END_FUNCTION_BLOCK

// POUs/Engineering/signal processing/SH_T
FUNCTION_BLOCK SH_T
VAR_INPUT
	IN : REAL;
	E : BOOL;
END_VAR
VAR_OUTPUT
	OUT : REAL;
END_VAR


(*
version 1.1	18. oct. 2008
programmer 	hugo
tested by	oscat

this sample and hold module samples an input while en is high.
during the high time of en the output follows in.
the out stays stable until the en goes high again.
*)

IF E THEN out := in; END_IF;



(* revision history
hm	1. sep. 2006	rev 1.0
	original version

hm	18. oct. 2008	rev 1.1
	changed input en to e for compatibility reasons

*)

END_FUNCTION_BLOCK

// POUs/Logic/gate logic/SHL1
FUNCTION SHL1 : DWORD
VAR_INPUT
	IN : DWORD;
	N : INT;
END_VAR
VAR CONSTANT
	temp : DWORD := 16#FFFF_FFFF;
END_VAR

(*
version 1.1	27 dec 2007
programmer 	hugo
tested by		tobias

SHL1 shifts N bits to the left filling the new bits with 1

*)

SHL1 := SHR(temp,32-N) OR SHL(IN,N);


(* revision history
hm	14.9.2007		rev 1.0
	original version

hm	27. dec 2007	rev 1.1
	changed code for better performance

*)

END_FUNCTION

// POUs/Logic/gate logic/SHR1
FUNCTION SHR1 : DWORD
VAR_INPUT
	IN : DWORD;
	N : INT;
END_VAR
VAR CONSTANT
	temp : DWORD := 16#FFFF_FFFF;
END_VAR

(*
version 1.1	27 dec 2007
programmer 	hugo
tested by		tobias

SHR1 shifts N bits to the right filling the new bits with 1

*)

SHR1 := SHL(temp,32-N) OR SHR(IN,N);

(* revision history
hm	14.9.2007		rev 1.0
	original version

hm	27. dec 2007	rev 1.1
	changed code for better performance

*)

END_FUNCTION

// POUs/Logic/FF edge triggered/SHR_4E
FUNCTION_BLOCK SHR_4E
VAR_INPUT
	SET : BOOL;
	D0: BOOL;
	CLK: BOOL;
	RST: BOOL;
END_VAR
VAR_OUTPUT
	Q0: BOOL;
	Q1: BOOL;
	Q2: BOOL;
	Q3: BOOL;
END_VAR
VAR
	trig : R_TRIG;
END_VAR

(*
version 1.1	25. oct. 2008
programmer 	hugo
tested by		tobias

4 bit shift register with reset

*)

(* trig.Q signals a rising edge on clk *)
trig(clk := clk);

IF set OR rst THEN
	Q0 := NOT rst;
	Q1 := Q0;
	Q2 := Q0;
	Q3 := Q0;
ELSIF trig.Q THEN
	Q3 := Q2;
	Q2 := Q1;
	Q1 := Q0;
	Q0 := D0;
END_IF;



(* revision history
hm	4. aug. 2006	rev 1.0
	original version

hm	25. oct. 2008	rev 1.1
	optimized code

*)

END_FUNCTION_BLOCK

// POUs/Logic/FF edge triggered/SHR_4UDE
FUNCTION_BLOCK SHR_4UDE
VAR_INPUT
	SET : BOOL;
	D0: BOOL;
	D3: BOOL;
	CLK: BOOL;
	DN : BOOL;
	RST: BOOL;

END_VAR
VAR_OUTPUT
	Q0: BOOL;
	Q1: BOOL;
	Q2: BOOL;
	Q3: BOOL;
END_VAR
VAR
	trig : R_TRIG;
END_VAR

(*
version 1.2	14. mar. 2009
programmer 	hugo
tested by		tobias

4 bit shift register with reset up / down direction input

*)

(* trig.Q signals a rising edge on clk *)
trig(clk := clk);

IF set OR rst THEN
	Q0 := NOT RST;
	Q1 := Q0;
	Q2 := Q0;
	Q3 := Q0;
ELSIF trig.Q THEN
	IF dn THEN
		Q0 := Q1;
		Q1 := Q2;
		Q2 := Q3;
		Q3 := D3;
	ELSE
		Q3 := Q2;
		Q2 := Q1;
		Q1 := Q0;
		Q0 := D0;
	END_IF;
END_IF;



(* revision history
hm	4. aug. 2006	rev 1.0
	original version

hm	25. oct. 2008	rev 1.1
	optimized code

hm	14. mar. 2009	rev 1.2
	removed double assignments

*)

END_FUNCTION_BLOCK

// POUs/Logic/FF edge triggered/SHR_8PLE
FUNCTION_BLOCK SHR_8PLE
VAR_INPUT
	Din : BOOL;
	Dload : BYTE;
	CLK: BOOL;
	UP: BOOL :=1;
	load : BOOL;
	RST: BOOL;
END_VAR
VAR_OUTPUT
	DOut: BOOL;
END_VAR
VAR
	edge : BOOL :=1;
	register : BYTE;
END_VAR

(*
version 1.0	4 aug 2006
programmer 	hugo
tested by	oscat

8 bit shift register with reset and parallel load
the register can shift up or down
it also has a serial input.
the Din input is on Bit0 for up shift and on bit 7 for down shift
the Dout output is on Bit7 for up shift and on bit 0 for down shift
paralle clock is performed clock synchron while a shift is performed first and then the register is reloaded


*)

(* flankenerkennung clk wird high und edge war high reset ist nicht aktiv und set ist nicht aktiv *)
IF CLK AND edge AND NOT rst THEN
	edge := FALSE;	(* flanke wurde erkannt und weitere flankenerkennung wird verhindert bis edge wieder true ist *)
	(* hier ist der code für das flankenevent *)
	IF UP THEN						(*shift up *)
		register := SHL(register,1);
		register.0 := Din;
		Dout := register.7;
	ELSE								(* shift down *);
		register := SHR(register,1);
		register.7 := Din;
		Dout := register.0;
	END_IF;
	IF load THEN							(* the byte on Din will be loaded if load = true *)
		register := Dload;
		IF up THEN Dout := register.7; ELSE Dout := register.0; END_IF;
	END_IF;
END_IF;
IF NOT clk THEN edge := TRUE; END_IF;	(* sobald clk wieder low wird warten auf nächste flanke *)
IF rst THEN									(* wenn reset aktiv dann ausgang rücksetzen *)
	register := 0;
	Dout := FALSE;
END_IF;

END_FUNCTION_BLOCK

// POUs/Logic/FF edge triggered/SHR_8UDE
FUNCTION_BLOCK SHR_8UDE
VAR_INPUT
	SET : BOOL;
	D0: BOOL;
	D7: BOOL;
	CLK: BOOL;
	DN : BOOL;
	RST: BOOL;
END_VAR
VAR_OUTPUT
	Q0: BOOL;
	Q1: BOOL;
	Q2: BOOL;
	Q3: BOOL;
	Q4: BOOL;
	Q5: BOOL;
	Q6: BOOL;
	Q7: BOOL;
END_VAR
VAR
	trig : R_TRIG;
END_VAR

(*
version 1.2	14. mar. 2009
programmer 	hugo
tested by		tobias

8 bit shift register with reset


*)

(* trig.Q signals a rising edge on clk *)
trig(clk := clk);

IF set OR rst THEN
	Q0 := NOT RST;
	Q1 := Q0;
	Q2 := Q0;
	Q3 := Q0;
	Q4 := Q0;
	Q5 := Q0;
	Q6 := Q0;
	Q7 := Q0;
ELSIF trig.Q THEN
	IF dn THEN
		Q0 := Q1;
		Q1 := Q2;
		Q2 := Q3;
		Q3 := Q4;
		Q4 := Q5;
		Q5 := Q6;
		Q6 := Q7;
		Q7 := D7;
	ELSE
		Q7 := Q6;
		Q6 := Q5;
		Q5 := Q4;
		Q4 := Q3;
		Q3 := Q2;
		Q2 := Q1;
		Q1 := Q0;
		Q0 := D0;
	END_IF;
END_IF;



(* revision history
hm	4. aug. 2006	rev 1.0
	original version

hm	25. oct. 2008	rev 1.1
	optimized code

hm	14. mar. 2009	rev 1.2
	removed double assignments

*)

END_FUNCTION_BLOCK

// POUs/Mathematical/SIGMOID
FUNCTION SIGMOID : REAL
VAR_INPUT
	X : REAL;
END_VAR


(*
version 1.2	10. mar. 2009
programmer 	hugo
tested by		tobias

this function calculates the sigmoid function

*)

IF X > 20.0 THEN
	SIGMOID := 1.0;
ELSIF x < -85.0 THEN
	SIGMOID := 0.0;
ELSE
	SIGMOID := 1.0 / (1.0 + EXP(-X));
END_IF;


(* revision history
hm	10.12.2007		rev 1.0
	original version

hm	11. mar. 2008		rev 1.1
	extended range of valid inputs to +inv / -inv

hm 10. mar. 2009		rev 1.2
	real constants updated to new systax using dot																																																																																																																																																																																																																																																																																																																																																																																																																																																																																																																																																																																																																																																																																																																																																																																																																																																																																																																																																																																																																																																											

*)

END_FUNCTION

// POUs/Mathematical/SIGN_I
FUNCTION SIGN_I : BOOL
VAR_INPUT
	IN : DINT;
END_VAR


(*
version 1.3	27. oct. 2008
programmer 	hugo
tested by	tobias

this function return true if the integer input is negative

*)

SIGN_I := in.31;

(* revision history
hm 3.3.2007	rev 1.1
	changed method of function for better compatibility to other systems

hm	1.12.2007	rev 1.2
	changed code to improve performance

hm	27. oct. 2008	rev 1.3
	changed type of input to dint

*)

END_FUNCTION

// POUs/Engineering/automation/SIGNAL_4
FUNCTION_BLOCK SIGNAL_4
VAR_INPUT
	IN1 : BOOL;
	IN2 : BOOL;
	IN3 : BOOL;
	IN4 : BOOL;
	TS : TIME;
END_VAR
VAR_INPUT CONSTANT
	S1 : BYTE := 2#1111_1111;
	S2 : BYTE := 2#1111_0000;
	S3 : BYTE := 2#1010_1010;
	S4 : BYTE := 2#1010_0000;
END_VAR
VAR_OUTPUT
	Q : BOOL;
END_VAR
VAR
	sig : SIGNAL;
END_VAR

(*
version 1.0	13 dec 2007
programmer 	hugo
tested by		tobias

this function generates one out of 4 signals specified by bit patterns S1 .. S4.
the selected pattern will be shifted with the step time TS.
In1 has higher priority then In2 which has higher priority then IN3 and in4 has the lowest priority.
ts defaults to 128 ms if not specified.
*)

(* an alarm is present read system time first *)
(* check if an alarm is present if yes set sig to the alarm pattern otherwise exit the routine *)
IF in1 THEN
	sig(in := TRUE, sig := s1, TS := TS);
ELSIF in2 THEN
	sig(in := TRUE, sig := s2, TS := TS);
ELSIF in3 THEN
	sig(in := TRUE, sig := s3, TS := TS);
ELSIF in4 THEN
	sig(in := TRUE, sig := s4, TS := TS);
ELSE
	sig(in := FALSE);
END_IF;

(* set the output *)
Q := sig.Q;


(* revision history
hm	13.12.2007		rev 1.0
	original version

*)

END_FUNCTION_BLOCK

// POUs/Mathematical/SINC
FUNCTION SINC : REAL
VAR_INPUT
	X : REAL;
END_VAR


(*
version 1.2	10. mar. 2009
programmer 	hugo
tested by		tobias

this function calculates the sinc function.

*)

IF X = 0.0 THEN
	SINC := 1.0;
ELSE
	SINC := SIN(x) / x;
END_IF;


(* revision histroy
hm	11. mar. 2008	rev 1.0
	original version

hm	1.12.2007	rev 1.1
	changed code to improove performance

hm 10. mar. 2009	rev 1.2
	real constants updated to new systax using dot																																																																																																																																																																																																																																																																																																																																																																																																																																																																																																																																																																																																																																																																																																																																																																																																																																																																																																																																																																																																																																																											

*)

END_FUNCTION

// POUs/Mathematical/Geometry/SPHERE_V
FUNCTION SPHERE_V : REAL
VAR_INPUT
	rx : REAL;
END_VAR


(*
version 1.2	22. feb 2008
programmer 	hugo
tested by		tobias

sphere_V calculates the Volume of a Sphere


*)

sphere_V := 4.188790205 * Rx * RX * RX;

(* revision histroy
hm	16. oct 2007	rev 1.0
	original version

hm	4. dec 2007		rev 1.1
	changed code for better performance

hm	22. feb 2008		rev 1.2
	changed code for better performance
*)

END_FUNCTION

// POUs/Engineering/automation/SRAMP
FUNCTION_BLOCK SRAMP
VAR_INPUT
	X : REAL;
	A_UP : REAL;
	A_DN :REAL;
	VU_MAX : REAL;
	VD_MAX : REAL;
	LIMIT_HIGH : REAL;
	LIMIT_LOW : REAL;
	RST : BOOL;
END_VAR
VAR_OUTPUT
	Y : REAL;
	V : REAL;
END_VAR
VAR
	cycle_time : TC_S;
	init: BOOL;
END_VAR


(*
	version 1.1	11. mar. 2009
	programmer 	hugo
	tested by		tobias

RAMPS generates output signal which are slew rate and acceleration controlled.

*)

(* read the system_time in microseconds *)
cycle_time();

(* assure range of inputs *)
A_up := MAX(0.0, A_UP);
A_dn := MIN(0.0, A_dn);
VU_max := MAX(0.0, VU_max);
VD_max := MIN(0.0, VD_MAX);

(* calculate the output offset *)
IF rst OR NOT init THEN
	init := TRUE;
	Y := 0.0;
	V := 0.0;
ELSIF X = Y THEN
	v := 0.0;
ELSIF X > Y THEN
	(* output is too low >> ramp up and brake at the end *)
	(* accelerate the speed and limit to vu_max *)
	v := MIN(v + A_UP * cycle_time.TC, vu_max);
	(* calculate the max speed to be able to brake and select the lowest *)
	v := MIN(SQRT((Y-X) * 2.0 * A_DN), v);
	(* calculate the output and obey limits *)
	y := LIMIT(limit_low, y + MIN(v * cycle_time.TC, X-Y), limit_high);
ELSIF X < Y THEN
	(* output is too high >> ramp dn and brake at the end *)
	(* accelerate the speed and limit to vd_max *)
	v := MAX(v + A_DN * cycle_time.TC, vd_max);
	(* calculate the max speed to be able to brake and select the lowest *)
	v := MAX(-SQRT((Y-X) * 2.0 * A_UP), v);
	(* calculate the output and obey limits *)
	y := LIMIT(limit_low, y + MAX(v * cycle_time.TC, X-Y), limit_high);
END_IF;


(* revision history
hm	13. mar. 2008	rev 1.0
	original version

hm	11. mar. 2009	rev 1.1
	real constants updated to new systax using dot																																																																																																																																																																																																																																																																																																																																																																																																																																																																																																																																																																																																																																																																																																																																																																																																																																																																																																																																																																																																																																																											

*)

END_FUNCTION_BLOCK

// POUs/Engineering/measurements/TC_S
FUNCTION_BLOCK TC_S

VAR_OUTPUT
	TC : REAL;
END_VAR
VAR
	init: BOOL;
	tx: DWORD;
	last: DWORD;
END_VAR

(*
	version 1.2	11. mar. 2009
	programmer 	hugo
	tested by		tobias

TC_S delivers the time it was last called on the output TC in seconds.

*)

(* read system timer *)
tx := T_PLC_US();

IF NOT init THEN
	init := TRUE;
	TC := 0.0;
ELSE
	tc := DWORD_TO_REAL(tx - last)*1.0E-6;
END_IF;
last := tx;

(* revision history
hm	13. mar. 2008	rev 1.0
	original version

hm	16. mar 2008	rev 1.1
	added type conversion to avoid warnings under codesys 3.0

hm	11. mar. 2009	rev 1.2
	changed real constants to use dot syntax

*)

END_FUNCTION_BLOCK

// POUs/Logic/memory/STACK_16
FUNCTION_BLOCK STACK_16
VAR_INPUT
	Din : DWORD;
	E : BOOL := TRUE;
	RD : BOOL;
	WD : BOOL;
	RST : BOOL;
END_VAR
VAR_OUTPUT
	Dout : DWORD;
	EMPTY : BOOL := TRUE;
	FULL : BOOL;
END_VAR
VAR
	stack : ARRAY[0..n] OF DWORD;
	pt : INT;
END_VAR
VAR CONSTANT
	n : INT := 15;	(* changing this value will chage the number of stored elements in the fifo *)
END_VAR


(*
version 2.0	25. jul 2009
programmer 	hugo
tested by		oscat

16 Dword STACK memory

*)

IF RST THEN
	(* asynchronous reset for the fifo *)
	pt := 0;
	EMPTY := TRUE;
	FULL := FALSE;
	Dout := 0;
ELSIF E THEN
	IF NOT EMPTY AND RD THEN
		(* read one element *)
		pt := pt - 1;
		Dout := stack[pt];
		EMPTY := pt = 0;
		FULL := FALSE;
	END_IF;
	IF NOT FULL AND WD THEN
		(* write one element *)
		stack[pt] := Din;
		pt := pt + 1;
		FULL := pt > n;
		EMPTY := FALSE;
	END_IF;
END_IF;


(* revision history
hm	4. aug. 2006	rev 1.0
	original version

hm	19. feb 2008	rev 1.1
	performance improvements

hm	17. oct. 2008	rev 1.2
	deleted unnecessary init with 0

hm	27. oct. 2008	rev 1.3
	optimized performance

hm	25. jul 2009	rev 2.0
	changed inputs to allow simultsaneous read and write
*)

END_FUNCTION_BLOCK

// POUs/Logic/memory/STACK_32
FUNCTION_BLOCK STACK_32
VAR_INPUT
	Din : DWORD;
	E : BOOL := TRUE;
	RD : BOOL;
	WD : BOOL;
	RST : BOOL;
END_VAR
VAR_OUTPUT
	Dout : DWORD;
	EMPTY : BOOL := TRUE;
	FULL : BOOL;
END_VAR
VAR
	stack : ARRAY[0..n] OF DWORD;
	pt : INT;
END_VAR
VAR CONSTANT
	n : INT := 31;	(* changing this value will chage the number of stored elements in the fifo *)
END_VAR


(*
version 2.0	25. jul 2009
programmer 	hugo
tested by		oscat

32 Dword STACK memory
*)

IF RST THEN
	(* asynchronous reset for the fifo *)
	pt := 0;
	EMPTY := TRUE;
	FULL := FALSE;
	Dout := 0;
ELSIF E THEN
	IF NOT EMPTY AND RD THEN
		(* read one element *)
		pt := pt - 1;
		Dout := stack[pt];
		EMPTY := pt = 0;
		FULL := FALSE;
	END_IF;
	IF NOT FULL AND WD THEN
		(* write one element *)
		stack[pt] := Din;
		pt := pt + 1;
		FULL := pt > n;
		EMPTY := FALSE;
	END_IF;
END_IF;


(* revision history
hm	4. aug. 2006	rev 1.0
	original version

hm	19. feb 2008	rev 1.1
	performance improvements

hm	17. oct. 2008	rev 1.2
	deleted unnecessary init with 0

ks	27. oct. 2008	rev 1.3
	optimized performance

hm	25. jul 2009	rev 2.0
	changed inputs to allow simultsaneous read and write

*)

END_FUNCTION_BLOCK

// POUs/Engineering/signal processing/STAIR
FUNCTION STAIR : REAL
VAR_INPUT
	X : REAL;
	D : REAL;
END_VAR


(*
version 1.4	10. mar. 2009
programmer 	oscat
tested by		tobias

the function stair converts an anlog input signal to a staircase like output.
D is the step width for the output signal.
if D = 0 then the output follows the input without a chage.
*)

IF D > 0.0 THEN
	STAIR := DINT_TO_REAL(REAL_TO_DINT(X / D)) * D;
ELSE
	STAIR := X;
END_IF;



(* revision history
hm	28 jan 2007		rev 1.0
	original version

hm	27 dec 2007		rev 1.1
	changed code for better performance

hm	6. jan 2008		rev 1.2
	further performance improvement

hm	26. oct. 2008		rev 1.3
	optimized code

hm	10. mar. 2009	rev 1.4
	real constants updated to new systax using dot

*)

END_FUNCTION

// POUs/Engineering/signal processing/STAIR2
FUNCTION_BLOCK STAIR2
VAR_INPUT
	X : REAL;
	D : REAL;
END_VAR
VAR_OUTPUT
	Y: REAL;
END_VAR


(*
version 1.4	10. mar. 2009
programmer 	hugo
tested by		oscat

the function stair2 converts an anlog input signal to a staircase like output.
D is the step width for the output signal. the output will use D as a hysteresis for a stairchange.
if D = 0 then the output follows the input without a chage.
*)

IF D > 0.0 THEN
	IF X >= Y + D OR X <= Y - D THEN Y := FLOOR(X/D) * D; END_IF;
ELSE
	Y := X;
END_IF;



(* revision history
hm	28 jan 2007		rev 1.0
	original version

hm	27. dec 2007	rev 1.1
	changed code for better performance

hm	30. jun. 2008	rev 1.2
	added type conversions to avoid warnings under codesys 3.0																																																																																																																																																																																																																																																											

ks	26. oct. 2008	rev 1.3
	improved code

hm	10. mar. 2009	rev 1.4
	real constants updated to new systax using dot

*)

END_FUNCTION_BLOCK

// POUs/Logic/FF pulse triggered/STORE_8
FUNCTION_BLOCK STORE_8
VAR_INPUT
	Set : BOOL;
	D0,D1, D2, D3, D4, D5, D6, D7 : BOOL;
	Clr : BOOL;
	Rst : BOOL;
END_VAR
VAR_OUTPUT
	Q0, Q1, Q2, Q3, Q4, Q5, Q6, Q7 : BOOL;
END_VAR
VAR
	edge: BOOL;
END_VAR

(*
version 1.2	14. mar. 2009
programmer 	hugo
tested by		oscat

Store_4 stores up to 4 boolean inputs until a reset is clearing the outputs.
the respective output is set with a true at the respective input and stays true until a reset is generated.
a set input is used to set all outputs true at the same time, independent of their inputs.
a clear input is used to reset only the lowest priority of the outputs one at a time.
the lowest priority is q3.

*)

IF rst OR set THEN
	q0 := NOT rst;
	q1 := q0;
	q2 := q0;
	q3 := q0;
	q4 := q0;
	q5 := q0;
	q6 := q0;
	q7 := q0;
ELSE
	IF D0 THEN Q0 := TRUE; END_IF;
	IF D1 THEN Q1 := TRUE; END_IF;
	IF D2 THEN Q2 := TRUE; END_IF;
	IF D3 THEN Q3 := TRUE; END_IF;
	IF D4 THEN Q4 := TRUE; END_IF;
	IF D5 THEN Q5 := TRUE; END_IF;
	IF D6 THEN Q6 := TRUE; END_IF;
	IF D7 THEN Q7 := TRUE; END_IF;

	IF clr AND NOT edge THEN
		IF q0 THEN q0 := FALSE;
		ELSIF q1 THEN q1 := FALSE;
		ELSIF q2 THEN q2 := FALSE;
		ELSIF q3 THEN q3 := FALSE;
		ELSIF q4 THEN q4 := FALSE;
		ELSIF q5 THEN q5 := FALSE;
		ELSIF q6 THEN q6 := FALSE;
		ELSE q7 := FALSE;
		END_IF;
	END_IF;
	edge := clr;
END_IF;


(* revision history
hm	25.12.2007	rev 1.0
	original version

hm	30. oct. 2008	rev 1.1
	optimized performance

hm	14. mar. 2009	rev 1.2
	removed double assignments

*)

END_FUNCTION_BLOCK

// POUs/Logic/gate logic/SWAP_BYTE
FUNCTION SWAP_BYTE : WORD
VAR_INPUT
	IN : WORD;
END_VAR


(*
version 1.0	4 feb 2008
programmer 	hugo
tested by		tobias

This function swaps the high and low byte of the word in.

*)

SWAP_BYTE := ROL(in,8);


(* revision history
hm		4. feb 2008	rev 1.0
	original version

*)

END_FUNCTION

// POUs/Logic/gate logic/SWAP_BYTE2
FUNCTION SWAP_BYTE2 : DWORD
VAR_INPUT
	IN : DWORD;
END_VAR


(*
version 1.0	4 feb 2008
programmer 	hugo
tested by		tobias

This function reverses the byte order in the dword.

*)

Swap_Byte2 := (ROR(in,8) AND 16#FF00FF00) OR (ROL(in,8) AND 16#00FF00FF);

(* revision history
hm		4. feb 2008	rev 1.0
	original version

*)

END_FUNCTION

// POUs/Mathematical/TANC
FUNCTION TANC : REAL
VAR_INPUT
	X : REAL;
END_VAR


(*
version 1.1	10. mar. 2009
programmer 	hugo
tested by		oscat

this function calculates the tanc function.

*)

IF X = 0.0 THEN
	TANC := 1.0;
ELSE
	TANC := TAN(x) / x;
END_IF;


(* revision histroy
hm	23. oct. 2008	rev 1.0
	original version

hm 10. mar. 2009	rev 1.1
	real constants updated to new systax using dot																																																																																																																																																																																																																																																																																																																																																																																																																																																																																																																																																																																																																																																																																																																																																																																																																																																																																																																																																																																																																																																											

*)

END_FUNCTION

// POUs/Mathematical/TANH
FUNCTION TANH : REAL
VAR_INPUT
	X : REAL;
END_VAR


(*
version 1.3	10. mar. 2009
programmer 	hugo
tested by		tobias

this function calculates the tangens hyperbolicus

*)

IF X > 20.0 THEN
	TANH := 1.0;
ELSIF X < -20.0 THEN
	TANH := -1.0;
ELSE
	TANH := 1.0 - 2.0 / (EXP(2.0 * x) + 1.0);
END_IF;


(* revision hisdtory
hm		12.1.2007		rev 1.0
	original version

hm		1.12.2007		rev 1.1
	changed code to improve performance

hm		10. mar 2008	rev 1.2
	corrected an error in formula
	extended range of valid inputs to +/- INV

hm 10. mar. 2009	rev 1.3
	real constants updated to new systax using dot																																																																																																																																																																																																																																																																																																																																																																																																																																																																																																																																																																																																																																																																																																																																																																																																																																																																																																																																																																																																																																																											

*)

END_FUNCTION

// POUs/Engineering/measurements/TC_MS
FUNCTION_BLOCK TC_MS

VAR_OUTPUT
	TC : DWORD;
END_VAR
VAR
	init: BOOL;
	tx: DWORD;
	last: DWORD;
END_VAR

(*
	version 1.0	13 mar 2008
	programmer 	hugo
	tested by		tobias

TC_MS delivers the time it was last called on the output TC in Milliseconds.

*)

(* read system timer *)
tx := T_PLC_MS();

IF NOT init THEN
	init := TRUE;
	TC := 0;
ELSE
	tc := tx - last;
END_IF;
last := tx;

(* revision history
hm		13. mar. 2008	rev 1.0
	original version

*)

END_FUNCTION_BLOCK

// POUs/Engineering/measurements/TC_US
FUNCTION_BLOCK TC_US

VAR_OUTPUT
	TC : DWORD;
END_VAR
VAR
	init: BOOL;
	tx: DWORD;
	last: DWORD;
END_VAR

(*
	version 1.0	13 mar 2008
	programmer 	hugo
	tested by		tobias

TC_US delivers the time it was last called on the output TC in Microseconds.

*)

(* read system timer *)
tx := T_PLC_US();

IF NOT init THEN
	init := TRUE;
	TC := 0;
ELSE
	tc := tx - last;
END_IF;
last := tx;

(* revision history
hm		13. mar. 2008	rev 1.0
	original version

*)

END_FUNCTION_BLOCK

// POUs/Engineering/sensor/TEMP_NI
FUNCTION TEMP_NI : REAL
VAR_INPUT
	Res : REAL;
	R0 : REAL;
END_VAR


(*
version 1.5	10. mar. 2009
programmer 	hugo
tested by		tobias

this function returns the temperature for a nickel sensor in a range from -60..+180 °C *)

TEMP_NI := (SQRT(0.30085225 - 2.66E-3 * (R0 - Res)) - 0.5485) * 751.8796992;


(* revision history

hm 24.1.2007		rev 1.1
	deleted unused variable A, B, C

hm 10.9.2007		rev 1.2
	changed accuracy to 0.02 degrees to improove performace

hm 17. 12 2007	rev 1.3
	improovements for better performance and higher accuracy

hm	6. jan 2008	rev 1.4
	further performance improvement

hm	10. mar. 2009	rev 1.5
	removed nested comments

*)

END_FUNCTION

// POUs/Engineering/sensor/TEMP_NTC
FUNCTION TEMP_NTC : REAL
VAR_INPUT
	RES : REAL;
	RN : REAL;
	B : REAL;
END_VAR


(*
version 1.1	11. mar. 2009
programmer 	hugo
tested by		tobias

this function returs the temperature for a NTC sensor for a range from 0..85 °C.
RN is the resistance at 25 °C and B is a constant for the given sensor.

*)

IF res > 0.0 THEN
	TEMP_NTC := B * 298.15 / (B + LN(RES / RN) * 298.15) -273.15;
END_IF;


(* revision history

hm 30. dec. 2008	rev 1.0
	original version

hm	11. mar. 2009	rev 1.1
	changed real constants to use dot syntax

*)

END_FUNCTION

// POUs/Engineering/sensor/TEMP_PT
FUNCTION TEMP_PT : REAL
VAR_INPUT
	Res : REAL;
	R0 : REAL;
END_VAR
VAR CONSTANT
	A : REAL := 3.9083E-3 ;
	B : REAL := -5.775E-7;
	accuracy : REAL := 0.01;
END_VAR
VAR
	step: REAL := 50.0;
	X: REAL;
	Y: REAL;
	t1: REAL;
	pt : POINTER TO DWORD;
END_VAR

(*
version 1.7	11. mar. 2009
programmer 	hugo
tested by		oscat

this function returs the temperature for a platinum sensor for a range from -200..+850 °C *)

X := A * R0;
Y := B * R0;
IF Res >= R0 THEN
	t1 := X * X - 4.0 * Y * (R0 - Res);
	IF t1 < 0.0 THEN
		TEMP_PT := 10000.0;
	ELSE
		TEMP_PT := (-X + SQRT(t1)) / (2.0 * Y);
	END_IF;
ELSE
	pt := ADR(step);
	(* since the formula cannot be solved this is a successive approximation *)
	TEMP_PT := -100.0;
	WHILE step > accuracy DO
		(* test if result greater or less *)
		IF RES_PT(TEMP_PT, R0) < res THEN TEMP_PT := TEMP_PT + step; ELSE TEMP_PT := TEMP_PT - step; END_IF;
		pt^ := pt^ - 8388608;  (* this is a super fast divide by 2 method for non floating point CPUs *)
		(* the alternative code: step := step * 0.5; *)
	END_WHILE;
END_IF;

(* revision history

rev 1.1 hm 24.1.2007	
	deleted unused variable C

rev 1.2 hm 10.9.2007
	reduced accuracy to 0.02 to shorten execution time

rev 1.3	hm	2. dec 2007
	changed code for better performance

rev	1.4	hm	23. dec 2007
	avoid a negative square root if input values are wrong

rev 1.5 hm	5. jan 2008
	replaced / 2 with * 0.5 for better performance

hm	31. oct. 2008	rev 1.6
	improved performance

hm	11. mar. 2009	rev 1.7
	changed real constants to use dot syntax

*)

END_FUNCTION

// POUs/Engineering/sensor/TEMP_SI
FUNCTION TEMP_SI : REAL
VAR_INPUT
	Res : REAL;
	RS : REAL;
	TS : REAL;
END_VAR


(*
version 1.5	10. mar. 2009
programmer 	hugo
tested by		tobias

this function returs the temperature for a silicon sensor for a range from -60..+180 °C
for example KTY10 RS at TS normally 25 °C
*)

TEMP_SI := (-7.64E-3 + SQRT(Res / RS * 6.64E-5 - 0.803E-5)) * 30120.48193 + TS;



(* revision history

hm 24.1.2007		rev 1.1
	the function would only work for TS = 25, now it works for other values of ts.

hm 10.9.2007		rev 1.2
	changed the function to use successive approcimation to avoid an error generated by a sqrt from a negative result.
	changed accuracy to 0.02 degrees to shorten execution time

hm 17. 12 2007	rev 1.3
	improovements for better performance

hm	6. jan 2008	rev 1.4
	further performance improvement

hm	10. mar. 2009	rev 1.5
	removed nested comments

*)

END_FUNCTION

// POUs/String/TICKER
FUNCTION_BLOCK TICKER

VAR_INPUT
	N : INT;
	PT : TIME;
END_VAR

VAR_IN_OUT
	Text : STRING(STRING_LENGTH);
END_VAR

VAR_OUTPUT
	Display : STRING(STRING_LENGTH);
END_VAR
VAR
	delay : TP;
	step : INT;
END_VAR

(*
version 1.2	29. mar. 2008
programmer 	hugo
tested by		tobias

Ticker sends a substring of text with length N every TD Milliseconds to generate a ticker. 

*)


(* generate next ticker when delay is low *)
IF N < LEN(text) THEN
	IF NOT delay.Q THEN
		(* increase step for next tick *)
		step := step + 1;
		IF step > LEN(text) THEN step := 1; END_IF;
		(* extract dispay from text *)
		display := MID(text, N, step);
		(* set delay timer for next tick *)
		delay(in := TRUE, PT := PT);
	ELSE;
		(* execute delay timer *)
		delay(in := FALSE);
	END_IF;
ELSE
	display := text;
END_IF;
(* revision history
hm	4. dec. 2007	rev 1.0
	original version

hm	15. dec. 2007	rev 1.1
	step now starts at 1 instaed of 0

hm	29. mar. 2008	rev 1.2
	changed STRING to STRING(STRING_LENGTH)
*)

END_FUNCTION_BLOCK

// POUs/Time&Date/TIMECHECK
FUNCTION TIMECHECK : BOOL
VAR_INPUT
	TD : TOD;
	START : TOD;
	STOP : TOD;
END_VAR


(*
version 1.0	19. jul. 2009
programmer 	oscat
tested by		oscat

this function retruns true if the daytime TD is between start and stop and returns true if so.
if you want to generate an event to span over midnight, start timemust be later than the stop time.

*)

IF stop < start THEN
	TIMECHECK := start <= TD OR TD < stop;
ELSE
	TIMECHECK := start <= TD AND TD < stop;
END_IF;



(* revision history
hm 19. jul. 2009	rev 1.0
	original release

*)

END_FUNCTION

// POUs/Logic/generators/TMIN
FUNCTION_BLOCK TMIN
VAR_INPUT
	IN : BOOL;
	PT : TIME;
END_VAR
VAR_OUTPUT
	Q : BOOL;
END_VAR
VAR
	pm : TP;
END_VAR

(*
version 1.0	21. jul. 2008
programmer 	hugo
tested by	oscat

Q of tMIN will follow IN except that it forces a minimum ontime for the output Q.

*)

pm(in := IN, PT := PT);
Q := IN OR pm.Q;


(* revision history
hm	21. jul. 2008	rev 1.0
	original version

*)

END_FUNCTION_BLOCK

// POUs/Logic/generators/TOF_1
FUNCTION_BLOCK TOF_1
VAR_INPUT
	IN : BOOL;
	PT : TIME;
	RST : BOOL;
END_VAR
VAR_OUTPUT
	Q : BOOL;
END_VAR
VAR
	tx : TIME;
	start : TIME;
END_VAR

(*
version 1.0	17. jul. 2008
programmer 	hugo
tested by	oscat

TOF_1 will extend a pulse on input in for PT seconds.
in addition the timer can be cleared asynchronously with rst.
TOF_1 is the same function as TOF from the standard LIB except the asynchronous reset input.

*)

(* read system timer *)
tx := DWORD_TO_TIME(T_PLC_MS());

IF RST THEN
	Q := FALSE;
ELSIF IN THEN
	Q := TRUE;
	start := tx;
ELSIF tx - start >= PT THEN
	Q := FALSE;
END_IF;




(* revision history
hm	17. jul. 2008	rev 1.0
	original version

*)

END_FUNCTION_BLOCK

// POUs/Logic/generators/TONOF
FUNCTION_BLOCK TONOF
VAR_INPUT
	IN : BOOL;
	  T_ON,T_OFF : TIME;
END_VAR
VAR_OUTPUT
	Q : BOOL;
END_VAR
VAR
   X : TON;
   old: BOOL;
   mode: BOOL;
END_VAR

(*
version 1.2	21. jul 2009
programmer 	hugo
tested by		tobias

TONOF generated a TON and TOF Delay for the Input N TON (T1) and TOF (T2) can be configured separately
*)

IF IN XOR old THEN
  X(IN := FALSE, PT := SEL(IN,T_OFF,T_ON));
  mode := IN;
  old := IN;
END_IF;
X(IN := TRUE);
IF X.Q THEN Q := mode;END_IF;

(* revision history
hm	10. dec 2007	rev 1.0
	original version

hm	17. sep. 2007	rev 1.1
	improved performance

hm	21. jul. 2009	rev 1.2
	fixed a timing probelm


*)

END_FUNCTION_BLOCK

// POUs/Logic/generators/TP_1
FUNCTION_BLOCK TP_1
VAR_INPUT
	IN : BOOL;
	PT : TIME;
	RST : BOOL;
END_VAR
VAR_OUTPUT
	Q : BOOL;
END_VAR
VAR
	tx : TIME;
	start : TIME;
	ix : BOOL;
END_VAR

(*
version 1.0	28. jun. 2008
programmer 	hugo
tested by		oscat

TP_1 generates a pulse every time it is calles with in := TRUE.
in addition the timer can be cleared asynchronously with rst.
the timer can be retriggered as often as necessary. it will count PT from the last trigger.

*)

(* read system timer *)
tx := DWORD_TO_TIME(T_PLC_MS());

IF RST THEN
	Q := FALSE;
ELSIF IN AND NOT ix THEN
	Q := TRUE;
	start := tx;
ELSIF tx - start >= PT THEN
	Q := FALSE;
END_IF;

ix:= IN;



(* revision history
hm	28. jun. 2008
	original version

*)

END_FUNCTION_BLOCK

// POUs/Mathematical/Geometry/TRIANGLE_A
FUNCTION TRIANGLE_A : REAL
VAR_INPUT
	S1 : REAL;
	A : REAL;
	S2 : REAL;
	S3 : REAL;
END_VAR


(*
version 1.2	10. mar. 2009
programmer 	hugo
tested by		tobias

triangle_A calculates the Area of a triangle.
if any input is 0 it will be neglected and the are will be calculated from eiter:
two sides and an angle (s1 and S2 and the angle A1) or 3 sides.


*)

IF A = 0.0 THEN
	TRIANGLE_A := SQRT((s1+s2+S3) * (s1+s2-S3) * (S2+S3-S1) * (S3+S1-S2)) * 0.25;
ELSE
	TRIANGLE_A := S1 * S2 * SIN(RAD(A)) * 0.5;
END_IF;

(* revision histroy
hm	16. oct 2007	rev 1.0
	original version

hm	22. feb 2008	rev 1.1
	improved performance

hm	10. mar. 2009	rev 1.2
	changed syntax of real constants to 0.0

*)

END_FUNCTION

// POUs/String/TRIM1
FUNCTION TRIM1 : STRING(STRING_LENGTH)
VAR_INPUT
	str : STRING(STRING_LENGTH);
END_VAR
VAR
	pos: INT;
END_VAR

(*
version 1.2	29. mar. 2008
programmer 	hugo
tested by		tobias

the function replaces all multiple blanks within a string by only one blank.
leading and ending blanks will be deleted

*)

TRIM1 := str;
REPEAT
	pos := FIND(trim1,'  ');
	IF pos > 0 THEN TRIM1 := REPLACE(TRIM1,' ',2,pos); END_IF;
UNTIL pos = 0	END_REPEAT;
(* beginning and ending blanks need to be stripped off *)
IF LEFT(trim1,1) = ' ' THEN trim1 := DELETE(trim1,1,1); END_IF;
IF RIGHT(trim1,1) = ' ' THEN trim1 := DELETE(trim1,1,LEN(trim1)); END_IF;


(* revision histroy
hm	4. feb. 2008    rev 1.0
	original release

hm	20. mar. 2008	rev 1.1
	avoid to call replace with pos = 0 because some systems will produce an error

hm	29. mar. 2008	rev 1.2
	changed STRING to STRING(STRING_LENGTH)
*)

END_FUNCTION

// POUs/String/TRIME
FUNCTION TRIME : STRING(string_length)
VAR_INPUT
	str : STRING(STRING_LENGTH);
END_VAR


(*
version 1.0	28. mar. 2008
programmer 	hugo
tested by	tobias

this function deletes all leading and ending blanks of a string.

*)

TRIME := str;
(* beginning blanks need to be stripped off *)
WHILE LEFT(TRIME,1) = ' ' DO
	TRIME := DELETE(TRIME,1,1);
END_WHILE;

(* ending blanks need to be stripped off *)
WHILE RIGHT(TRIME,1) = ' ' DO
	TRIME := DELETE(TRIME,1,LEN(TRIME));
END_WHILE;


(* revision histroy
hm	28. mar. 2008	rev 1.0
	original release

*)

END_FUNCTION

// POUs/Engineering/automation/TUNE
FUNCTION_BLOCK TUNE
VAR_INPUT
	SET : BOOL;
	SU, SD : BOOL;
	RST : BOOL;
END_VAR
VAR_INPUT CONSTANT
	SS : REAL := 0.1;
	Limit_L : REAL;
	LIMIT_H : REAL := 100.0;
	RST_val : REAL;
	SET_val : REAL := 100.0;
	T1 : TIME := T#500ms;
	T2 : TIME := T#2s;
	S1 : REAL := 2.0;
	S2 : REAL := 10.0;
END_VAR
VAR_OUTPUT
	Y : REAL;
END_VAR
VAR
	tx : DWORD;
	start, start2 : DWORD;
	state : INT;
	in : BOOL;
	step : REAL;
	SPEED : REAL;
	Y_start : REAL;
	Y_start2: REAL;
END_VAR

(*
version 1.2	11. mar. 2009
programmer 	hugo
tested by		tobias

tune generates an output signal which is set by input switches.
up to 4 switsches can be used to tune the signal up or down.

*)

(* read system time *)
tx := T_PLC_MS();

IF rst THEN
	Y := RST_val;
	state := 0;
ELSIF set THEN
	Y := SET_val;
	state := 0;
ELSIF state > 0 THEN
	(* key has been pushed state machine operating *)
	(* first read the correct input *)
	IF state = 1 THEN
		(* step up *)
		in := su;
	ELSE
		(* step down *)
		in := sd;
	END_IF;
	(* check for single step operation *)
	IF NOT in AND tx - start <= TIME_TO_DWORD(T1) THEN
		Y := Y_start + step;
		state := 0;
	(* check if fast ramp needs to be generated *)
	ELSIF in AND tx - start >= TIME_TO_DWORD(T2) THEN
		Y := Y_start2 + DWORD_TO_REAL(tx - start2) * s2 / speed;
	(* check if slow ramp needs to be generated *)
	ELSIF in AND tx - start >= TIME_TO_DWORD(T1) THEN
		Y := Y_start + DWORD_TO_REAL(tx - start - TIME_TO_DWORD(T1)) * S1 / speed;
		start2 := tx;
		Y_start2 := Y;
	ELSIF NOT in THEN
		state := 0;
	END_IF;
ELSIF su THEN
	(* slow step up *)
	state := 1;
	start := tx;
	step := ss;
	speed := 1000.0;
	Y_start := Y;
ELSIF sd THEN
	(* slow step down *)
	state := 2;
	start := tx;
	step := -ss;
	speed := -1000.0;
	Y_start := Y;
END_IF;

(* make sure output does not exceed limits *)
Y := LIMIT(LIMIT_L, Y, LIMIT_H);

(* revision history
hm	3.11.2007		rev 1.0
	original version

hm	16. mar. 2008	rev 1.1
	added type conversions to avoid warnings under codesys 3.0

hm	11. mar. 2009	rev 1.2
	real constants updated to new systax using dot																																																																																																																																																																																																																																																																																																																																																																																																																																																																																																																																																																																																																																																																																																																																																																																																																																																																																																																																																																																																																																																											

*)

END_FUNCTION_BLOCK

// POUs/Engineering/automation/TUNE2
FUNCTION_BLOCK TUNE2
VAR_INPUT
	SET : BOOL;
	SU, SD : BOOL;
	FU, FD : BOOL;
	RST : BOOL;
END_VAR
VAR_INPUT CONSTANT
	SS : REAL := 0.1;
	FS : REAL := 5.0;
	Limit_L : REAL;
	LIMIT_H : REAL := 100.0;
	RST_val : REAL;
	SET_val : REAL := 100.0;
	TR : TIME := T#500ms;
	S1 : REAL := 2.0;
	S2 : REAL := 10.0;
END_VAR
VAR_OUTPUT
	Y : REAL;
END_VAR
VAR
	tx : DWORD;
	start : DWORD;
	state : INT;
	in : BOOL;
	step : REAL;
	SPEED : REAL;
	Y_start : REAL;
END_VAR

(*
version 1.2	11. mar. 2009
programmer 	hugo
tested by		tobias

tune2 generates an output signal which is set by input switches.
up to 4 switsches can be used to tune the signal up or down.

*)

(* read system time *)
tx := T_PLC_MS();

IF rst THEN
	Y := RST_val;
	state := 0;
ELSIF set THEN
	Y := SET_val;
	state := 0;
ELSIF state > 0 THEN
	(* key has been pushed state machine operating *)
	(* first read the correct input *)
	CASE state OF
		1 :	(* slow up *)
			in := su;
		2 :	(* slow down *)
			in := sd;
		3 :	(* fast up *)
			in := fu;
		4 :	(* fast down *)
			in := fd;
	END_CASE;
	(* check for single step operation *)
	IF NOT in AND tx - start <= TIME_TO_DWORD(TR) THEN
		Y := Y_start + step;
		state := 0;
	(* check if ramp needs to be generated *)
	ELSIF in AND tx - start >= TIME_TO_DWORD(TR) THEN
		Y := Y_start + DWORD_TO_REAL(tx - start - TIME_TO_DWORD(TR)) * speed;
	ELSIF NOT in THEN
		state := 0;
	END_IF;
ELSIF su THEN
	(* slow step up *)
	state := 1;
	start := tx;
	step := ss;
	speed := s1 * 1.0E-3;
	Y_start := Y;
ELSIF sd THEN
	(* slow step down *)
	state := 2;
	start := tx;
	step := -ss;
	speed := -s1 * 1.0E-3;
	Y_start := Y;
ELSIF fu THEN
	(* fast step up *)
	state := 3;
	start := tx;
	step := fs;
	speed := s2 * 1.0E-3;
	y_start := Y;
ELSIF fd THEN
	(* fast step down *)
	state := 4;
	start := tx;
	step := -fs;
	speed := -s2 * 1.0E-3;
	y_start := Y;
END_IF;

(* make sure output does not exceed limits *)
Y := LIMIT(LIMIT_L, Y, LIMIT_H);

(* revision history
hm	3.11.2007		rev 1.0
	original version

hm	16. 3. 2008	rev 1.1
	added type conversions to avoid warnings in codesys 3.0
	improved performance

hm	11. mar. 2009	rev 1.2
	real constants updated to new systax using dot																																																																																																																																																																																																																																																																																																																																																																																																																																																																																																																																																																																																																																																																																																																																																																																																																																																																																																																																																																																																																																																											

*)

END_FUNCTION_BLOCK

// POUs/Mathematical/Vektormathematik/V3_ABS
FUNCTION V3_ABS : REAL
VAR_INPUT
	A : Vector_3;
END_VAR


(*
version 1.0	11 dec 2007
programmer 	hugo
tested by		tobias

this function calculates the length of a vectors in a 3 dimensional space

*)

V3_ABS := SQRT(A.X * A.X + A.Y * A.Y + A.Z * A.Z);


(* revision history
hm		11 dec 2007	rev 1.0
	original version

*)

END_FUNCTION

// POUs/Mathematical/Vektormathematik/V3_ADD
FUNCTION V3_ADD : vector_3
VAR_INPUT
	A : Vector_3;
	B : Vector_3;
END_VAR


(*
version 1.0	11 dec 2007
programmer 	hugo
tested by		tobias

this function adds two vectors in a 3 dimensional space

*)

V3_ADD.X := A.X + B.X;
V3_ADD.Y := A.Y + B.Y;
V3_ADD.Z := A.Z + B.Z;



(* revision history
hm		11 dec 2007	rev 1.0
	original version

*)

END_FUNCTION

// POUs/Mathematical/Vektormathematik/V3_ANG
FUNCTION V3_ANG : REAL
VAR_INPUT
	A : Vector_3;
	B : Vector_3;
END_VAR
VAR
	d : REAL;
END_VAR

(*
version 1.1	10. mar. 2009
programmer 	hugo
tested by		tobias

this function calculates the angle between two vectors in a 3 dimensional space

*)

d := V3_ABS(A) * V3_ABS(B);
IF d > 0 THEN
	V3_ANG := ACOS(LIMIT(-1.0, V3_DPRO(A, B) / d,1.0));
END_IF;

(* revision history
hm	11. dec. 2007	rev 1.0
	original version

hm	10. mar. 2009	rev 1.1
	changed syntax of real constants to 0.0

*)

END_FUNCTION

// POUs/Mathematical/Vektormathematik/V3_DPRO
FUNCTION V3_DPRO : REAL
VAR_INPUT
	A : Vector_3;
	B : Vector_3;
END_VAR


(*
version 1.0	11 dec 2007
programmer 	hugo
tested by		tobias

this function calculates the dot product of two vectors in 3 dimensional space

*)

V3_DPRO := A.X * B.X + A.Y * B.Y + A.Z * B.Z;


(* revision history
hm		11 dec 2007	rev 1.0
	original version

*)

END_FUNCTION

// POUs/Mathematical/Vektormathematik/V3_NORM
FUNCTION V3_NORM : vector_3
VAR_INPUT
	A : Vector_3;
END_VAR
VAR
	la: REAL;
END_VAR

(*
version 1.1	10. mar. 2009
programmer 	hugo
tested by		tobias

this function generates a vectors with absolute length 1 from a vector A in a 3 dimensional space

*)

la := V3_ABS(A);
IF la > 0.0 THEN
	V3_NORM := V3_SMUL(A, 1.0 / la);
END_IF;

(* revision history
hm	11 dec 2007	rev 1.0
	original version

hm	10. mar. 2009	rev 1.1
	changed syntax of real constants to 0.0

*)

END_FUNCTION

// POUs/Mathematical/Vektormathematik/V3_SMUL
FUNCTION V3_SMUL : vector_3
VAR_INPUT
	A : Vector_3;
	M : REAL;
END_VAR


(*
version 1.0	11 dec 2007
programmer 	hugo
tested by		tobias

this function multiplies a vectors in a 3 dimensional space with a skalar M

*)

V3_SMUL.X := A.X * M;
V3_SMUL.Y := A.Y * M;
V3_SMUL.Z := A.Z * M;



(* revision history
hm		11 dec 2007	rev 1.0
	original version

*)

END_FUNCTION

// POUs/Mathematical/Vektormathematik/V3_NUL
FUNCTION V3_NUL : BOOL
VAR_INPUT
	A : Vector_3;
END_VAR


(*
version 1.1	10. mar. 2009
programmer 	hugo
tested by		tobias

this function checks if a vectors in a null Vector

*)

V3_NUL := A.X = 0.0 AND A.Y = 0.0 AND A.Z = 0.0;



(* revision history
hm	12 dec 2007	rev 1.0
	original version

hm	10. mar. 2009	rev 1.1
	changed syntax of real constants to 0.0

*)

END_FUNCTION

// POUs/Mathematical/Vektormathematik/V3_PAR
FUNCTION V3_PAR : BOOL
VAR_INPUT
	A : Vector_3;
	B : Vector_3;
END_VAR


(*
version 1.1	10. mar. 2009
programmer 	hugo
tested by		tobias

this function checks if two vectors in a 3 dimensional space are parallel.
which means the two vectors have the same direction

*)

V3_PAR := V3_ABS(V3_XPRO(A, B)) = 0.0;



(* revision history
hm	11 dec 2007	rev 1.0
	original version

hm	10. mar. 2009	rev 1.1
	changed syntax of real constants to 0.0

*)

END_FUNCTION

// POUs/Mathematical/Vektormathematik/V3_XPRO
FUNCTION V3_XPRO : vector_3
VAR_INPUT
	A : Vector_3;
	B : Vector_3;
END_VAR


(*
version 1.0	11 dec 2007
programmer 	hugo
tested by		tobias

this function adds two vectors in a 3 dimensional space

*)

V3_XPRO.X := A.Y * B.Z - A.Z * B.Y;
V3_XPRO.Y := A.Z * B.X - A.X * B.Z;
V3_XPRO.Z := A.X * B.Y - A.Y * B.X;



(* revision history
hm		11 dec 2007	rev 1.0
	original version

*)

END_FUNCTION

// POUs/Mathematical/Vektormathematik/V3_REV
FUNCTION V3_REV : vector_3
VAR_INPUT
	A : Vector_3;
END_VAR


(*
version 1.0	11 dec 2007
programmer 	hugo
tested by		tobias

this function reverses a vector in a 3 dimensional space

*)

V3_REV.X := -A.X;
V3_REV.Y := -A.Y;
V3_REV.Z := -A.Z;



(* revision history
hm		11 dec 2007	rev 1.0
	original version

*)

END_FUNCTION

// POUs/Mathematical/Vektormathematik/V3_SUB
FUNCTION V3_SUB : vector_3
VAR_INPUT
	A : Vector_3;
	B : Vector_3;
END_VAR


(*
version 1.0	11 dec 2007
programmer 	hugo
tested by		tobias

this function subtracts two vectors in a 3 dimensional space
V3_SUB = A - B

*)

V3_SUB.X := A.X - B.X;
V3_SUB.Y := A.Y - B.Y;
V3_SUB.Z := A.Z - B.Z;



(* revision history
hm		11 dec 2007	rev 1.0
	original version

*)

END_FUNCTION

// POUs/Mathematical/Vektormathematik/V3_XANG
FUNCTION V3_XANG : REAL
VAR_INPUT
	A : Vector_3;
END_VAR
VAR
	la: REAL;
END_VAR

(*
version 1.1	10. mar. 2009
programmer 	hugo
tested by		tobias

this function calculates the angle between the X-axis and a vectors in a 3 dimensional space

*)

la := V3_ABS(a);
IF la > 0.0 THEN
	V3_XANG := ACOS(A.X / la);
END_IF;

(* revision history
hm	11 dec 2007	rev 1.0
	original version

hm	10. mar. 2009	rev 1.1
	changed syntax of real constants to 0.0

*)

END_FUNCTION

// POUs/Mathematical/Vektormathematik/V3_YANG
FUNCTION V3_YANG : REAL
VAR_INPUT
	A : Vector_3;
END_VAR
VAR
	la: REAL;
END_VAR

(*
version 1.1	10. mar. 2009
programmer 	hugo
tested by		tobias

this function calculates the angle between the Y-axis and a vectors in a 3 dimensional space

*)

la := V3_ABS(a);
IF la > 0.0 THEN
	V3_YANG := ACOS(A.Y / la);
END_IF;

(* revision history
hm	11 dec 2007	rev 1.0
	original version

hm	10. mar. 2009	rev 1.1
	changed syntax of real constants to 0.0

*)

END_FUNCTION

// POUs/Mathematical/Vektormathematik/V3_ZANG
FUNCTION V3_ZANG : REAL
VAR_INPUT
	A : Vector_3;
END_VAR
VAR
	la: REAL;
END_VAR

(*
version 1.1	10. mar. 2009
programmer 	hugo
tested by		tobias

this function calculates the angle between the Z-axis and a vectors in a 3 dimensional space

*)

la := V3_ABS(a);
IF la > 0.0 THEN
	V3_ZANG := ACOS(A.Z / la);
END_IF;

(* revision history
hm	11 dec 2007	rev 1.0
	original version

hm	10. mar. 2009	rev 1.1
	changed syntax of real constants to 0.0

*)

END_FUNCTION

// POUs/Mathematical/WINDOW2
FUNCTION WINDOW2 : BOOL
VAR_INPUT
	LOW : REAL;
	IN : REAL;
	HIGH : REAL;
END_VAR


(*
	version 1.0	31 oct 2007
	programmer 	hugo
	tested BY	tobias

this checks a signal if the signal is between the upper and lower limit including the two limits
*)

WINDOW2 := IN >= LOW AND IN <= HIGH;


(* revision history
hm	31.10.2007	rev 1.0
	original version

*)

END_FUNCTION

// POUs/Logic/gate logic/WORD_OF_BYTE
FUNCTION WORD_OF_BYTE : WORD
VAR_INPUT
	B1 : BYTE;
	B0 : BYTE;
END_VAR


(*
version 1.4	18. jul. 2009
programmer 	hugo
tested by		tobias

this function creates a word from 2 individual bytes

*)

WORD_OF_BYTE := SHL(BYTE_TO_WORD(B1),8) OR BYTE_TO_WORD(B0);

(* revision history
hm	24. jan 2007	rev 1.0
	original version

hm	2. jan 2008	rev 1.1
	improved performance

hm	19. feb 2008	rev 1.2
	replaced and with or for better compatibility

hm	23. apr. 2008	rev 1.3
	reverse order of inputs to be more logical

hm	18. jul. 2009	rev 1.4
	added type conversions for compatibility reasons

*)

END_FUNCTION

// POUs/Logic/gate logic/WORD_OF_DWORD
FUNCTION WORD_OF_DWORD : WORD
VAR_INPUT
	in : DWORD;
	N : BYTE;
END_VAR


(*
version 1.2	30. oct. 2008
programmer 	hugo
tested by	oscat

this function extracts a single word from the nth position from right (right is lowest byte)
the lower word (starting with Bit0 from in) is selected with N=0.
*)

WORD_OF_DWORD := DWORD_TO_WORD(SHR(in,SHL(n,4)));

(* revision history
hm	17. jan 2007	rev 1.0
	original version

hm	2. jan 2008		rev 1.1
	improved performance

hm	30. oct. 2008	rev 1.2
	improved performance
*)

END_FUNCTION

// POUs/Engineering/signal processing/WORD_TO_RANGE
FUNCTION WORD_TO_RANGE : REAL
VAR_INPUT
	X : WORD;
	low : REAL;
	high : REAL;
END_VAR


(*
version 1.1	10. mar. 2009
programmer 	hugo
tested by		tobias

Word_to_Range converts a Byte into a real between low and high.

*)

WORD_TO_RANGE := (high - low) * WORD_TO_REAL(X) * 0.00001525902189669640 + low;


(* revision history
hm	9. jan 2008	rev 1.0
	original version

hm	10. mar. 2009	rev 1.1
	improved code
*)

END_FUNCTION

// POUs/Time&Date/YEAR_END
FUNCTION YEAR_END : DATE
VAR_INPUT
	y : INT;
END_VAR


(*
version 1.1	24. jan. 2011
programmer 	hugo
tested by	oscat

returs the date of december 31st for the given year  
the function works for dates from 1970 - 2099 

*)

YEAR_END := DWORD_TO_DATE(SHR(INT_TO_DWORD(y) * 1461 - 2876712, 2) * 86400);



(* revision history
hm	15. jun. 2008	rev 1.0
	original version

hm	24. jan 2011	rev 1.1
	improved performance
*)

END_FUNCTION

// POUs/String/LREAL_TO_STRF
FUNCTION LREAL_TO_STRF : STRING(40)
VAR_INPUT
	IN : LREAL;
	N : INT;
	D : STRING(1);
END_VAR
VAR
	O: LREAL;
	i: INT;
END_VAR

(*
version 1.8	2. jan 2012
programmer 	hugo
tested by	oscat

Real_to_strf converts a Real to a fixed length String.
the string will be filles with zeroes to achieve the fixed length N after the decimal separator.
the input parameter specifies the decimal separator to be used in the output string.

*)

(* LIMIT N to 0 .. 17 *)
N := LIMIT(0,N,17);
(* round the input to N digits and convert to string *)
O := ABS(in) * EXP10(N);
LREAL_TO_STRF := LINT_TO_STRING(LREAL_TO_LINT(O));
(* add zeroes in front to make sure string is at least 17 digits long *)
FOR i := LEN(LREAL_TO_STRF) TO N DO LREAL_TO_STRF := CONCAT('0', LREAL_TO_STRF); END_FOR;
(* add a dot if n > 0 *)
IF n > 0 THEN LREAL_TO_STRF := INSERT(LREAL_TO_STRF, D, LEN(LREAL_TO_STRF) - N); END_IF;
(* add a minus sign if in is negative *)
IF in < 0 THEN LREAL_TO_STRF := CONCAT('-', LREAL_TO_STRF); END_IF;


(* revision history
hm	26 jan 2007	rev 1.0
	original version

hm	20. nov. 2007	rev 1.1
	when N=0 ther will be no dot at the end of the string.

hm	15. dec. 2007	rev 1.2
	changed code for better performance

hm	4. mar. 2008	rev 1.3
	result is now rounded instead of trunc

hm	20. mar. 2008	rev 1.4
	changed trunc to real_to_dint because trunc was generating wrong values on wago 842

hm	29. mar. 2008	rev 1.5
	changed STRING to STRING(20)

hm	4. apr. 2008	rev 1.6
	added variable O to avoid an error uner CoDeSys SP PLCWinNT V2.4

hm	27. feb. 2009	rev 1.7
	added a missing zero for IN < 1

hm 2. jan 2012	rev 1.8
	added input parameter D to specify decimal separator
	
hm 10.10.2017 rev1.8
	added LREAL support
*)

END_FUNCTION
